{attribute 'GeneratedUsingTerminal: EL4014-0000-0018'}
{attribute addProperty BoxType "EL4014-0000-0018"}
{attribute addProperty Description "EL4014 4Ch. Ana. Output 0-20mA, 12bit"}
{attribute addProperty Physics "KK"}
{attribute addProperty Id "AO_Output_Channel_1AT %Q*AO_Output_Channel_BA7EBB7C2AO_Output_Channel_2AT %Q*AO_Output_Channel_BA7EBB7C2AO_Output_Channel_3AT %Q*AO_Output_Channel_BA7EBB7C2AO_Output_Channel_4AT %Q*AO_Output_Channel_BA7EBB7C2WcStateAT %I*WcState_0B2B16F91InfoDataAT %I*InfoData_32EB74EA10"}
{attribute addProperty CRC "365406740"}
{attribute addProperty Size "19"}
TYPE EL4014_15C7AA14 EXTENDS EtcSlaveTerminalBase_947E5A46 :
STRUCT
	{attribute addProperty Name "AO_Output_Channel_1"}
	AO_Output_Channel_1 : AO_Output_Channel_BA7EBB7C;
	{attribute addProperty Name "AO_Output_Channel_2"}
	AO_Output_Channel_2 : AO_Output_Channel_BA7EBB7C;
	{attribute addProperty Name "AO_Output_Channel_3"}
	AO_Output_Channel_3 : AO_Output_Channel_BA7EBB7C;
	{attribute addProperty Name "AO_Output_Channel_4"}
	AO_Output_Channel_4 : AO_Output_Channel_BA7EBB7C;
	{attribute addProperty Name "WcState"}
	WcState : WcState_0B2B16F9;
	{attribute addProperty Name "InfoData"}
	InfoData : InfoData_32EB74EA;
END_STRUCT
END_TYPE

(* stored: Version 1.2.0.0, ProductVersion 3.1.4024.11
   DUT EL4014_15C7AA14: Id {85137da0-534c-4c37-b86a-32cfe5455b1a} *)
